// LS Electric XG5000 project: 동남83
// PLC NewPLC
// module base 0 slot 0: 입출력 모듈:XBC-DN/DP14E (DC 24V 입력 8점, 트랜지스터 출력 6점)

PROGRAM NewProgram (task: 스캔 프로그램)

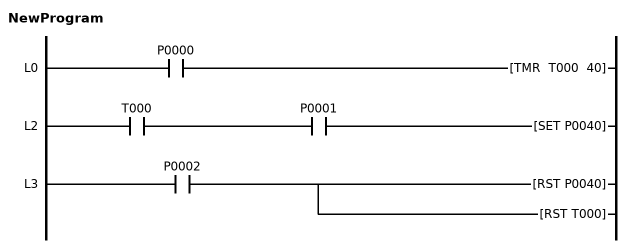
; L0
LOAD      P0000
TMR       T000 40
; L2
LOAD      T000
AND       P0001
SET       P0040
; L3
LOAD      P0002
RST       P0040
RST       T000